{attribute addProperty BoxType "EL5021-0000-0016"}
{attribute addProperty Id "StatusAT %I*Status_500944311621Counter_valueAT %I*UDINT32417Latch_valueAT %I*UDINT32418"}
{attribute addProperty CRC "872269726"}
{attribute addProperty SizeInBites "80"}
{attribute addProperty SizeInBytes "10"}
TYPE ENC_Status_33FDC79E :
STRUCT
	{attribute addProperty Name "Status"}
	Status AT %I* : Status_50094431;
	{attribute addProperty Name "Counter_value"}
	Counter_value AT %I* : UDINT;
	{attribute addProperty Name "Latch_value"}
	Latch_value AT %I* : UDINT;
END_STRUCT
END_TYPE

(* stored: Version 1.2.0.0, ProductVersion 3.1.4024.9
   DUT ENC_Status_33FDC79E: Id {60da303c-8cc9-4775-92bb-5fb9975251f1} *)
